% RSLogix 500 project I2P JOB 17 - MYAH.RSS, saved by version 10.00.00.00 %
PROJECT "UNTITLED"    % processor: Bul.1763 MicroLogix 1100 Series B %

PROGRAM FILES
  LAD 2   5 rungs

DATA FILES
  O0 OUTPUT  4 elements
  I1 INPUT  6 elements
  S2 STATUS  66 elements
  B3 BINARY  1 elements
  T4 TIMER  1 elements
  C5 COUNTER  1 elements
  R6 CONTROL  1 elements
  N7 INTEGER  1 elements
  F8 FLOAT  1 elements

LADDER 2
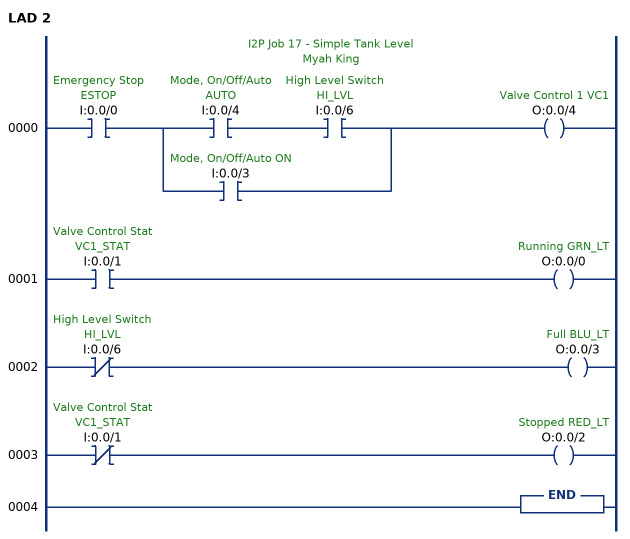
% Rung: 0 %
% I2P Job 17 - Simple Tank Level
% Myah King %
SOR XIC I:0.0/0 BST XIC I:0.0/4 XIC I:0.0/6 NXB XIC I:0.0/3 BND OTE O:0.0/4 EOR
%   I:0.0/0  ESTOP  "Emergency Stop" %
%   I:0.0/4  AUTO  "Mode, On/Off/Auto" %
%   I:0.0/6  HI_LVL  "High Level Switch" %
%   I:0.0/3  ON  "Mode, On/Off/Auto" %
%   O:0.0/4  VC1  "Valve Control 1" %
% Rung: 1 %
SOR XIC I:0.0/1 OTE O:0.0/0 EOR
%   I:0.0/1  VC1_STAT  "Valve Control Stat" %
%   O:0.0/0  GRN_LT  "Running" %
% Rung: 2 %
SOR XIO I:0.0/6 OTE O:0.0/3 EOR
%   I:0.0/6  HI_LVL  "High Level Switch" %
%   O:0.0/3  BLU_LT  "Full" %
% Rung: 3 %
SOR XIO I:0.0/1 OTE O:0.0/2 EOR
%   I:0.0/1  VC1_STAT  "Valve Control Stat" %
%   O:0.0/2  RED_LT  "Stopped" %
% Rung: 4 %
SOR END EOR

OTHER DOCUMENTED ADDRESSES
  I:0.0/5  OFF_AUTO  "Off or Auto"
  O:0.0/1  YLW_LT  "Auto"
